FUNCTION_BLOCK FB_StationDismantling
VAR_INPUT
	Enable:				BOOL;
	System:				REFERENCE TO ST_System;
	Station:			REFERENCE TO ST_SystemStation;
	Error:				REFERENCE TO ST_Error;
	Setting:			REFERENCE TO ST_Setting;
	Recipe:				REFERENCE TO ST_Recipe;	
	Parameter:			REFERENCE TO ST_StationDismantling;	
END_VAR
VAR_OUTPUT
END_VAR
VAR
	_i:					INT;
	_arrTon:		    ARRAY[0..20] OF TON;
	_arrFbErrorTag:		ARRAY[0..20] OF FB_ErrorTag;
	_arrState:			ARRAY[0..20] OF BOOL;
	_bOpenLockTemp:		BOOL;
	_bResetLockTemp:	BOOL;
	_stHandshake:		ST_StationDismantlingHandshake;
END_VAR

A_Home();
A_Auto();

ACTION A_Auto:
CASE Station.iStepNow OF
	1000:
		Station.arrInfo[E_Language.Chinese]:="初始化完成 等待启动";
		IF  Enable THEN
			Station.iStepNext:=1101;
		END_IF
	1101:
		Station.arrInfo[E_Language.Chinese]:="判断是否有料";
		Parameter.eState:=E_StationState.Busy;
		IF NOT Parameter.bClose AND NOT Parameter.bPalletCheck2 THEN
			Station.iStepNext:=1201;
		END_IF
	1201:
		Station.arrInfo[E_Language.Chinese]:="请求放料";
		Parameter.eState:=E_StationState.Load;
		Station.iStepNext:=1301;
	1301:
		Parameter.stHandshake.bRequestLineLoad_D:=TRUE;
		IF Parameter.stHandshake.bResponseDismantling_D THEN
			Parameter.eState:=E_StationState.Busy;
			Station.iStepNext:=1401;
		END_IF
	1401:
		Station.arrInfo[E_Language.Chinese]:="等待产品流入";
		IF Parameter.bPalletCheck2 THEN
			Station.iStepNext:=1501;
		END_IF
	1501:
		Station.arrInfo[E_Language.Chinese]:="复位放料请求";
		Parameter.stHandshake.bRequestLineLoad_D:=FALSE;
		IF NOT Parameter.stHandshake.bResponseDismantling_D THEN
			Station.iStepNext:=1601;
		END_IF
	1601:
		Station.arrInfo[E_Language.Chinese]:="等待产品到位";
		IF Parameter.bPalletCheck2 THEN
			Station.iStepNext:=1701;
		END_IF
	1701:
		Station.arrInfo[E_Language.Chinese]:="顶升气缸上升 阻挡气缸缩回";
		_bOpenLockTemp:=FALSE;
		_arrState[0]:=Parameter.fbLift.M_WorkRequest() ;
		_arrState[1]:=Parameter.fbPrevent.M_HomeRequest();
		IF _arrState[0] AND _arrState[1]THEN
			Station.iStepNext:=1801;
		END_IF
	1801:
		Station.arrInfo[E_Language.Chinese]:="载具解锁";
		IF M_OpenLock() THEN
			Station.iStepNext:=1901;
		END_IF
	1901:
		Station.arrInfo[E_Language.Chinese]:="校平气缸伸出";
		IF M_StandardWork() THEN
			Station.iStepNext:=2001;
		END_IF
	2001:
		Station.arrInfo[E_Language.Chinese]:="请求取UC";
		Parameter.stHandshake.bRequestUc:=TRUE;
		IF Parameter.stHandshake.bResponseDismantling_Uc THEN
			Station.iStepNext:=2201;
		END_IF
	2201:
		Parameter.stHandshake.bRequestUc:=FALSE;
		IF NOT Parameter.stHandshake.bResponseDismantling_Uc THEN
			Station.iStepNext:=2301;
		END_IF
	2301:
		Station.arrInfo[E_Language.Chinese]:="校平气缸缩回";
		_bResetLockTemp:=FALSE;
		IF M_StandardHome() THEN
			Station.iStepNext:=2401;
		END_IF
	2401:
		Station.arrInfo[E_Language.Chinese]:="载具复位";
		IF M_ResetLock() THEN
			Station.iStepNext:=2501;
		END_IF
	2501:
		Station.arrInfo[E_Language.Chinese]:="判断下工装站是否屏蔽";
		IF NOT  Parameter.bCloseUnloadElevator THEN
			Station.iStepNext:=2551;
		ELSIF Parameter.fbLift.M_HomeRequest() THEN
			Station.iStepNext:=2801;
		END_IF
	2551:
		Station.arrInfo[E_Language.Chinese]:="请求下工装";
		Parameter.stHandshake.bRequestElevator:=TRUE;
		IF Parameter.stHandshake.bResponseDismantling_E THEN
			Station.iStepNext:=2601;
		END_IF
	2601:
		Station.arrInfo[E_Language.Chinese]:="顶升气缸下降";
		IF Parameter.fbLift.M_HomeRequest() THEN
			Station.iStepNext:=2701;
		END_IF
	2701:
		Station.arrInfo[E_Language.Chinese]:="复位请求";
		Parameter.stHandshake.bRequestElevator:=FALSE;
		IF NOT Parameter.stHandshake.bResponseDismantling_E THEN
			Station.iStepNext:=2801;
		END_IF
	2801:
		Station.arrInfo[E_Language.Chinese]:="等待产品流出";
		IF NOT Parameter.bPalletCheck1 AND NOT Parameter.bPalletCheck2 AND NOT Parameter.bPalletCheck3 THEN
			Station.iStepNext:=2901;
		END_IF
	2901:
		Station.arrInfo[E_Language.Chinese]:="阻挡气缸伸出";
		IF  Parameter.fbPrevent.M_WorkRequest() THEN
			Station.iStepNext:=1101;
		END_IF
END_CASE
END_ACTION

ACTION A_Home:
CASE Station.iStepNow OF
	0:
		Station.arrInfo[E_Language.Chinese]:="等待初始化";
		Parameter.stHandshake:=_stHandshake;
		Parameter.eState:=E_StationState.Done;
		Station.iStepNext:=SEL(Enable,1000,100);
	100:
		Station.arrInfo[E_Language.Chinese]:="阻挡气缸伸出";
		IF Parameter.fbPrevent.M_WorkRequest() THEN
			Station.iStepNext:=200;
		END_IF
	200:
		Station.arrInfo[E_Language.Chinese]:="侧推气缸缩回";
		IF M_LateralHome() THEN
			Station.iStepNext:=300;
		END_IF
	300:
		Station.arrInfo[E_Language.Chinese]:="旋转气缸复位";
		IF Parameter.fbRotate.M_HomeRequest() THEN
			Station.iStepNext:=400;
		END_IF
	400:
		Station.arrInfo[E_Language.Chinese]:="校平气缸缩回";
		IF M_StandardHome() THEN
			Station.iStepNext:=500;
		END_IF
	500:
		Station.arrInfo[E_Language.Chinese]:="顶升气缸缩回";
		IF Parameter.fbLift.M_HomeRequest() THEN
			Station.iStepNext:=1000;
		END_IF
END_CASE
END_ACTION

METHOD M_LateralHome : BOOL
VAR_INPUT
END_VAR
VAR
	_temp:			ARRAY[0..10] OF BOOL;
END_VAR
CASE Recipe.eMachineType OF
	E_MachineType.LH311,E_MachineType.RH311:
		M_LateralHome:=Parameter.fbLateral1.M_HomeRequest();
	E_MachineType.LH353,E_MachineType.RH353:
		_temp[0]:=Parameter.fbLateral1.M_HomeRequest();
		_temp[1]:=Parameter.fbLateral2.M_HomeRequest();
		M_LateralHome:=_temp[0] AND _temp[1];
	E_MachineType.LH367,E_MachineType.RH367:
		_temp[0]:=Parameter.fbLateral1.M_HomeRequest();
		_temp[1]:=Parameter.fbLateral2.M_HomeRequest();
		M_LateralHome:=_temp[0] AND _temp[1];
	E_MachineType.LH201,E_MachineType.RH201:
		_temp[0]:=Parameter.fbLateral1.M_HomeRequest();
		_temp[1]:=Parameter.fbLateral2.M_HomeRequest();
		M_LateralHome:=_temp[0] AND _temp[1];
	E_MachineType.LH069,E_MachineType.RH069:
		_temp[0]:=Parameter.fbLateral1.M_HomeRequest();
		_temp[1]:=Parameter.fbLateral2.M_HomeRequest();
		M_LateralHome:=_temp[0] AND _temp[1];
	E_MachineType.LH373,E_MachineType.RH373:
		M_LateralHome:=Parameter.fbLateral1.M_HomeRequest();
END_CASE
END_METHOD

METHOD M_LateralWork : BOOL
VAR_INPUT
END_VAR

VAR
	_temp: array[0..10] of bool;
END_VAR
CASE Recipe.eMachineType OF
	E_MachineType.LH311,E_MachineType.RH311:
		M_LateralWork:=Parameter.fbLateral1.M_WorkRequest();
	E_MachineType.LH353,E_MachineType.RH353:
		_temp[0]:=Parameter.fbLateral1.M_WorkRequest();
		_temp[1]:=Parameter.fbLateral2.M_WorkRequest();
		M_LateralWork:=_temp[0] AND _temp[1];
	E_MachineType.LH367,E_MachineType.RH367:
		_temp[0]:=Parameter.fbLateral1.M_WorkRequest();
		_temp[1]:=Parameter.fbLateral2.M_WorkRequest();
		M_LateralWork:=_temp[0] AND _temp[1];
	E_MachineType.LH201,E_MachineType.RH201:
		_temp[0]:=Parameter.fbLateral1.M_WorkRequest();
		_temp[1]:=Parameter.fbLateral2.M_WorkRequest();
		M_LateralWork:=_temp[0] AND _temp[1];
	E_MachineType.LH069,E_MachineType.RH069:
		_temp[0]:=Parameter.fbLateral1.M_WorkRequest();
		_temp[1]:=Parameter.fbLateral2.M_WorkRequest();
		M_LateralWork:=_temp[0] AND _temp[1];
	E_MachineType.LH373,E_MachineType.RH373:
		M_LateralWork:=Parameter.fbLateral1.M_WorkRequest();
END_CASE
END_METHOD

METHOD M_OpenLock : BOOL
VAR_INPUT
END_VAR
IF Recipe.eMachineType=E_MachineType.LH311 OR Recipe.eMachineType=E_MachineType.RH311 THEN
	IF M_LateralWork() THEN
		M_OpenLock:=Parameter.fbRotate.M_WorkRequest();
	END_IF
ELSE
	IF NOT _bOpenLockTemp THEN
		IF M_LateralWork() THEN
			_bOpenLockTemp:=Parameter.fbRotate.M_WorkRequest();
		END_IF
	ELSE
		CASE  Recipe.eMachineType OF
			E_MachineType.LH201,E_MachineType.RH201:
				M_OpenLock:=Parameter.fbLateral2.M_HomeRequest();
			ELSE
				M_OpenLock:=M_LateralHome();
		END_CASE
	END_IF
END_IF
END_METHOD

METHOD M_ResetLock : BOOL
VAR_INPUT
END_VAR
IF Recipe.eMachineType=E_MachineType.LH311 OR Recipe.eMachineType=E_MachineType.RH311 THEN
	IF M_LateralHome() THEN
		M_ResetLock:=Parameter.fbRotate.M_HomeRequest();;
	END_IF
ELSE
	IF NOT _bResetLockTemp THEN
		IF Parameter.fbLateral1.M_WorkRequest() THEN
			_bResetLockTemp:=Parameter.fbRotate.M_HomeRequest();
		END_IF
	ELSE
		M_ResetLock:=Parameter.fbLateral1.M_HomeRequest();
	END_IF
END_IF
END_METHOD

METHOD M_StandardHome : BOOL
VAR_INPUT
END_VAR
VAR
	_temp:			ARRAY[0..10] OF BOOL;
END_VAR
CASE Recipe.eMachineType OF
	E_MachineType.LH311,E_MachineType.RH311:
		_temp[0]:=Parameter.fbStandard1.M_HomeRequest();
		_temp[1]:=Parameter.fbStandard2.M_HomeRequest();
		M_StandardHome:=_temp[0] AND _temp[1];
	E_MachineType.LH353,E_MachineType.RH353:
		M_StandardHome:=Parameter.fbStandard1.M_HomeRequest();
	E_MachineType.LH367,E_MachineType.RH367:
		M_StandardHome:=Parameter.fbStandard1.M_HomeRequest();
	E_MachineType.LH201,E_MachineType.RH201:
		M_StandardHome:=TRUE;
	E_MachineType.LH069,E_MachineType.RH069:
		M_StandardHome:=TRUE;
	E_MachineType.LH373,E_MachineType.RH373:
		M_StandardHome:=Parameter.fbStandard1.M_HomeRequest();
END_CASE
END_METHOD

METHOD M_StandardWork : BOOL
VAR_INPUT
END_VAR

VAR
	_temp: array[0..10] of bool;
END_VAR
CASE Recipe.eMachineType OF
	E_MachineType.LH311,E_MachineType.RH311:
		_temp[0]:=Parameter.fbStandard1.M_WorkRequest();
		_temp[1]:=Parameter.fbStandard2.M_WorkRequest();
		M_StandardWork:=_temp[0] AND _temp[1];
	E_MachineType.LH353,E_MachineType.RH353:
		M_StandardWork:=Parameter.fbStandard1.M_WorkRequest();
	E_MachineType.LH367,E_MachineType.RH367:
		M_StandardWork:=Parameter.fbStandard1.M_WorkRequest();
	E_MachineType.LH201,E_MachineType.RH201:
		M_StandardWork:=TRUE;
	E_MachineType.LH069,E_MachineType.RH069:
		M_StandardWork:=TRUE;
	E_MachineType.LH373,E_MachineType.RH373:
		M_StandardWork:=TRUE;//Parameter.fbStandard1.M_WorkRequest();
END_CASE
END_METHOD

END_FUNCTION_BLOCK

(* stored: Version 1.1.0.1, ProductVersion 3.1.4024.3
   POU FB_StationDismantling: Id {a1d9aa93-cb9b-4363-9924-ff669d3c1f5e}, SpecialFunc None
   Action A_Auto: Id {dec06b43-b120-45f8-a55c-c24959594709}
   Action A_Home: Id {90e646ee-b30c-4cb8-a7d1-4bdf1d23fb1e}
   Method M_LateralHome: Id {cd2b8726-2fc4-40c0-9dcb-89fdc8100078}
   Method M_LateralWork: Id {6ed579ac-728a-4ab9-820b-430eb7174114}
   Method M_OpenLock: Id {04a3adc7-531b-498b-8990-e0e022908dce}
   Method M_ResetLock: Id {ae361eed-a379-4e59-ad4f-f639d9a12f80}
   Method M_StandardHome: Id {52a5c25a-bd78-4a64-99bf-f5691526a479}
   Method M_StandardWork: Id {1ca86bad-8d4c-45f1-8041-3fd933d3111a} *)
